INTERFACE ITcoRobotics EXTENDS __System.IQueryInterface

METHOD StartAtMain : TcoCore.ITcoTaskStatus
END_METHOD

METHOD StartMotorsAndProgram : TcoCore.ITcoTaskStatus
END_METHOD

METHOD StartMovements : TcoCore.ITcoTaskStatus
VAR_INPUT
	inData : TcoRoboticsMovementsParams;
END_VAR
END_METHOD

METHOD StopMovements : TcoCore.ITcoTaskStatus
VAR_INPUT
	inStopType : eTcoRoboticsStopType;
END_VAR
END_METHOD

METHOD StopMovementsAndProgram : TcoCore.ITcoTaskStatus
VAR_INPUT
	inStopType : eTcoRoboticsStopType;
END_VAR
END_METHOD

END_INTERFACE

(* stored: Version 1.1.0.1, ProductVersion 3.1.4024.12
   Itf ITcoRobotics: Id {57e4b936-bbfb-0eb5-372b-c0d667db345a}
   Folder Operations: Id {d8109b4c-19cd-0811-29f7-671663a0afa6}
   Method StartAtMain: Id {bc65f8ac-592f-0a2b-0415-1514fa61fa09}
   Method StartMotorsAndProgram: Id {f97f4746-dc86-05f2-25d6-03a7baaf43f9}
   Method StartMovements: Id {bf62d065-423a-059f-2635-b3395a365bf0}
   Method StopMovements: Id {4ab91db4-3107-074c-3b82-d32f9b392c09}
   Method StopMovementsAndProgram: Id {9427d102-9495-0c02-0bb7-83a6e19acc2a} *)
